FUNCTION TryConvert_LREAL_TO_LREAL : BOOL
VAR_INPUT
	in : LREAL;
	out : REFERENCE TO LREAL;
END_VAR

out := in;
TryConvert_LREAL_TO_LREAL := TRUE;

END_FUNCTION

(* stored: Version 1.1.0.1, ProductVersion 3.1.4024.12
   POU TryConvert_LREAL_TO_LREAL: Id {2b8f777d-672c-47a7-b5d4-da5b6e3fe40c}, SpecialFunc None *)
